Fanuc KAREL source: CA0035.KL

PROGRAM CA0035
%STACKSIZE=65535
%PRIORITY=65535
%NOLOCKGROUP
TYPE
T=STRUCTURE
A : INTEGER
B : REAL
ENDSTRUCTURE
VAR
G : INTEGER
I : INTEGER
R : REAL
B : BOOLEAN
S : STRING[16]
AI : ARRAY[2] OF INTEGER
AR : ARRAY[2] OF REAL
ST : T
P : XYZWPR
V : VECTOR
ROUTINE F(P1 : INTEGER; P2 : REAL; P3 : BOOLEAN; P4 : STRING; P5 : INTEGER; P6 : REAL; P7 : BOOLEAN; P8 : STRING; P9 : INTEGER; P10 : REAL; P11 : BOOLEAN; P12 : STRING) FROM CA0035
ROUTINE F
BEGIN
G=(G + 1)
END F
BEGIN
G=0
I=1
R=2.5
B=TRUE
S='A'
AI[1]=3
AR[1]=4.5
-- UNSAFE_SOURCE_IR line 42: ST.A = 5
-- UNSAFE_SOURCE_IR line 43: ST.B = 6.5
F(I,R,B,S,I,R,B,S,I,R,B,S)
END CA0035
